// TIA Portal V20 export
TYPE "type_emRelations_em8_cmStatus"
// stored: Access Published, Namespace Unit1
   STRUCT
      HipotThicknessSafetyPin : "LBC_typeDigitalSignalControlNode";
      HipotThicknessJRDetect : "LBC_typeDigitalSignalControlNode";
      ThicknessAxisZ : "LBC_typeAxis64PosControlNode";
      HipotThicknessStageLiftFrontUpDown : "LBC_typeTwoWayActuatorControlNode";
      HipotThicknessStageLiftRearUpDown : "LBC_typeTwoWayActuatorControlNode";
      HipotTabContactorBwdFwd : "LBC_typeTwoWayActuatorControlNode";
      HipotTabContactorLeftOpenClose : "LBC_typeTwoWayActuatorControlNode";
      HipotTabContactorRightOpenClose : "LBC_typeTwoWayActuatorControlNode";
      HipotThicknessStageLiftAllUpDown : "LBC_typeTwoWayActuatorControlNode";
      HipotThicknessServoPress : "LER_typeServoPressControlNode";
      ThicknessControl : "LER_typeThicknessControlNode";
      HipotControl : "LER_typeHipotControlNodes";
   END_STRUCT;
END_TYPE
